Staubli VAL3: aLight2.pgx

public program aLight2(num nValue (dimensions=1))
begin
  aioSet(aLight2,nValue)
end
